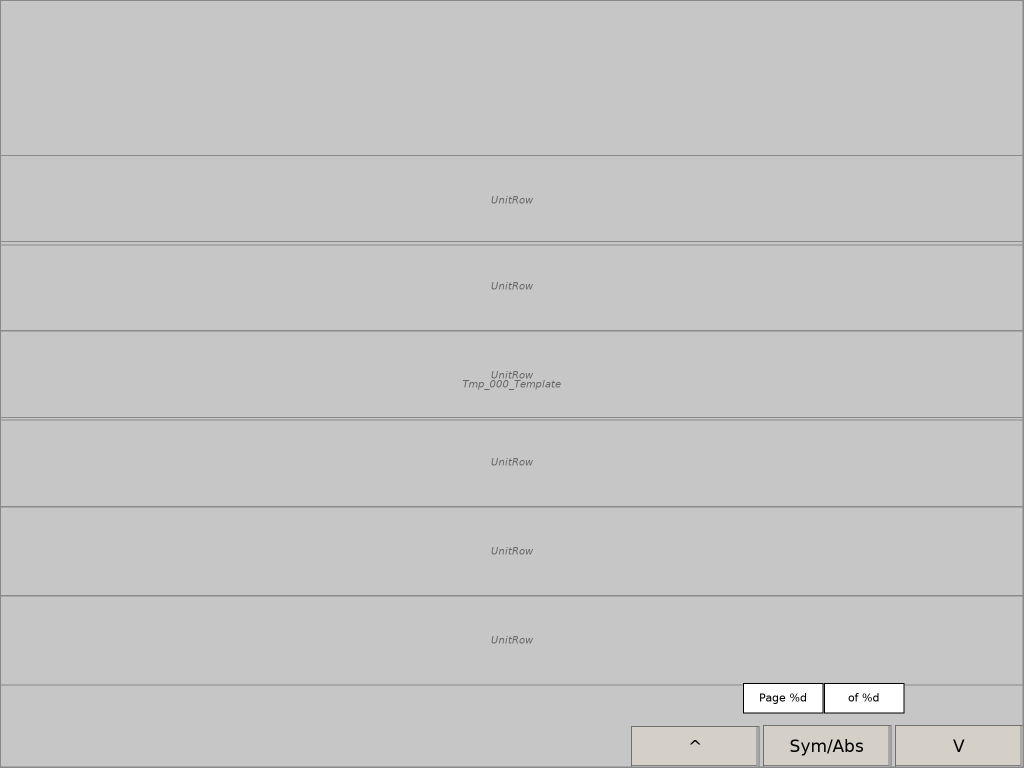
VISUALIZATION Unt_401_Units  // 1024x768
    Frame (0,0 1024x768)
        shows Tmp_000_Template(header := gHMIData.hmiHeader)
    Frame (0,155 1024x90)
        shows UnitRow(MotionRowInstanceSingle := gHMIUnits.gUnitRows.gMotionRow1, MotionRowButtonsSingle := gHMIUnits.gUnitButtons.gMotionRow1btn)
    Frame (0,241 1024x90)
        shows UnitRow(MotionRowInstanceSingle := gHMIUnits.gUnitRows.gMotionRow2, MotionRowButtonsSingle := gHMIUnits.gUnitButtons.gMotionRow2btn)
    Frame (0,330 1024x90)
        shows UnitRow(MotionRowInstanceSingle := gHMIUnits.gUnitRows.gMotionRow3, MotionRowButtonsSingle := gHMIUnits.gUnitButtons.gMotionRow3btn)
    Frame (0,417 1024x90)
        shows UnitRow(MotionRowInstanceSingle := gHMIUnits.gUnitRows.gMotionRow4, MotionRowButtonsSingle := gHMIUnits.gUnitButtons.gMotionRow4btn)
    Frame (0,506 1024x90)
        shows UnitRow(MotionRowInstanceSingle := gHMIUnits.gUnitRows.gMotionRow5, MotionRowButtonsSingle := gHMIUnits.gUnitButtons.gMotionRow5btn)
    Frame (0,595 1024x90)
        shows UnitRow(MotionRowInstanceSingle := gHMIUnits.gUnitRows.gMotionRow6, MotionRowButtonsSingle := gHMIUnits.gUnitButtons.gMotionRow6btn)
    Button (763,725 128x42), "Sym/Abs", colour toggle: gHMIButtons.btnAbsMode
        toggle gHMIButtons.btnAbsMode
    Button (631,726 128x41), "^"
        tap gHMIButtons.btnPrevPage
    Button (895,725 128x42), "V"
        tap gHMIButtons.btnNextPage
    Rectangle (743,683 80x30), "Page %d", text variable: gHMIData.gActivePageNumber
    Rectangle (824,683 80x30), "of %d", text variable: gHMIData.gMaxPageNumber
END_VISUALIZATION

(* stored: Version 1.1.0.1, ProductVersion 3.1.4024.11
   Visu Unt_401_Units: Id {1dd174fc-f423-007e-2b97-dad29a8ddd28} *)
